PROGRAM MathHelper
VAR
	_Random : DRAND;
END_VAR

METHOD ConvertDegreesToRadians : LREAL
VAR_INPUT
	degrees : LREAL;
END_VAR
ConvertDegreesToRadians := degrees * PI / 180;
END_METHOD

METHOD ConvertRadiansToDegrees : LREAL
VAR_INPUT
	radiand : LREAL;
END_VAR
ConvertRadiansToDegrees := radiand * 180 / PI;
END_METHOD

METHOD GetRandomValue : LREAL
VAR_INPUT
	seed : INT;
END_VAR
_Random(Seed := seed, Num => GetRandomValue);
END_METHOD

METHOD GetRandomWithDispersion : LREAL
VAR_INPUT
	baseValue : LREAL;
	dispersion : LREAL;	
END_VAR
GetRandomWithDispersion := baseValue - dispersion + (dispersion * 2 * MathHelper.GetRandomValue(0));
END_METHOD

METHOD GetRandomWithDispersionEx : LREAL
VAR_INPUT
	minValue : LREAL;
	baseValue : LREAL;
	maxValue : LREAL;
	dispersion : LREAL;	
END_VAR
GetRandomWithDispersionEx := baseValue - dispersion + (dispersion * 2 * MathHelper.GetRandomValue(0));

IF GetRandomWithDispersionEx < minValue THEN
	GetRandomWithDispersionEx := minValue;
ELSIF GetRandomWithDispersionEx > maxValue THEN
	GetRandomWithDispersionEx := maxValue;
END_IF
END_METHOD

METHOD Truncate : LREAL
VAR_INPUT
	value : LREAL;
	precission : BYTE;
END_VAR
VAR 
	i : INT;
	factor : LREAL := 1;
END_VAR
FOR i := 1 TO precission DO
	factor := factor * 10;
END_FOR

Truncate := TO_LREAL(TRUNC(value * factor)) / factor;
END_METHOD

END_PROGRAM

(* stored: Version 1.1.0.1
   POU MathHelper: Id {a7efcd16-5417-4251-b582-b89de7d35241}, SpecialFunc None
   Method ConvertDegreesToRadians: Id {a1cc6396-945d-4511-874b-e949879872ed}
   Method ConvertRadiansToDegrees: Id {2430e7d9-3523-44e4-8fc2-7240cac52474}
   Method GetRandomValue: Id {d36ecec8-180d-459b-b59c-dfd7219a70ef}
   Method GetRandomWithDispersion: Id {6de37dc6-155b-4776-bf24-269532044c36}
   Method GetRandomWithDispersionEx: Id {19d7d84f-24f3-412d-8955-cd454d1deaa8}
   Method Truncate: Id {78443544-2fdf-461c-8dde-3cbf14a580ad} *)
